// TIA Portal project "ton_ve_aa_4motorkontrolu" (V18)

(* hardware
DEVICE "S7-1200 station_1"  S7-1200 Station
   slot 0: "Rack_0"  S7-1200 Rack  Rack  V1.0
   slot 1: "PLC_1"  CPU 1214C AC/DC/Rly  6ES7 214-1BG40-0XB0  V4.6
*)

// ===== PLC "PLC_1"  CPU 1214C AC/DC/Rly =====

VAR_GLOBAL   // PLC tag table "Default tag table"
   "STOP" AT %I0.0 : Bool;
   "START" AT %I0.1 : Bool;
   "AA_1" AT %I0.2 : Bool;
   "AA_2" AT %I0.3 : Bool;
   "M1" AT %Q0.0 : Bool;
   "M2" AT %Q0.1 : Bool;
   "M3" AT %Q0.2 : Bool;
   "M4" AT %Q0.3 : Bool;
END_VAR

// folder: System blocks/Program resources

DATA_BLOCK "T1"   // DB1
{ S7_Optimized_Access := 'TRUE' }
AUTHOR : Simatic
FAMILY : IEC
NAME : IEC_TMR
VERSION : 1.0
// stored: InstanceOfName IEC_TIMER
"IEC_TIMER"
BEGIN
END_DATA_BLOCK

// folder: (top level)

ORGANIZATION_BLOCK "Main"   // OB1, LAD, ProgramCycle
TITLE = "Main Program Sweep (Cycle)"
{ S7_Optimized_Access := 'TRUE' }
VERSION : 0.1
   VAR_INPUT
      Initial_Call : Bool;   // Initial call of this OB
      Remanence : Bool;   // =True, if remanent data are available
   END_VAR
BEGIN

REGION Network 1
   // BİR MAKİNE TEZGAHINDA 4 ADET MOTOR ÇALIŞTIRILACAKTIR. STARTA BASILDIĞINDA 1 VE 3SÜREKLİ ÇALIŞACAK , HER İKİ MOTORADAN HERHANGİ BİRİSİNİN AŞIRI AKIM RÖLESİ ATTIĞINDA ONLARIN YERİNE 2 VE 4 NUMARALI MOTORLAR DEVREYE GİRECEKTİR. 2 VE 4 DEVREYE GİRDİĞİNDE BİRLİKTE 20SN ÇALILTIKTAN SONRA SİSTEM TAMAMIYLA DURACAKTIR. AYRICA STOP BUTONU HERHANGİ BİR ANDA SİSTEMİ DURDURABİLMEKTEDİR.
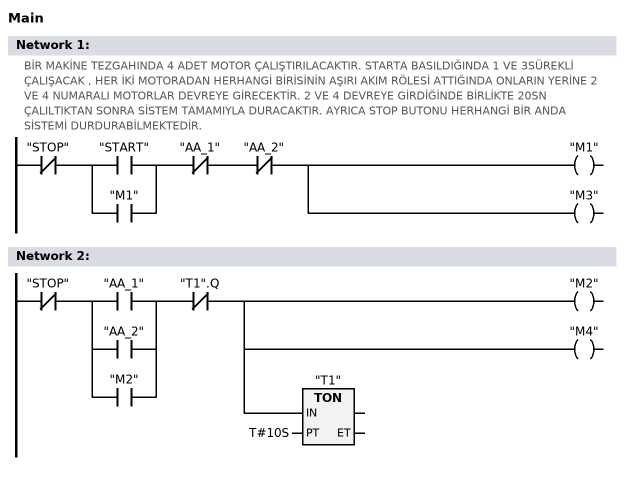
   RUNG wire#powerrail
      I_Contact( "STOP" )
      wire#w1
      Contact( "START" )
      wire#w2
      I_Contact( "AA_1" )
      I_Contact( "AA_2" )
      wire#w3
      Coil( "M1" )
   END_RUNG
   RUNG wire#w1
      Contact( "M1" )
   END_RUNG wire#w2
   RUNG wire#w3
      Coil( "M3" )
   END_RUNG
   // the same network as SCL:
   "M1" := NOT "STOP" AND ("START" OR "M1") AND NOT "AA_1" AND NOT "AA_2";
   "M3" := "M1";
END_REGION

REGION Network 2
   "M2" := NOT "STOP" AND ("AA_1" OR "AA_2" OR "M2") AND NOT "T1".Q;
   "M4" := "M2";
   "T1".TON(IN := "M2", PT := T#10S);
END_REGION
END_ORGANIZATION_BLOCK